// Mitsubishi GX Works2 project: PLC 특수기능 (연산 결과 반전)   PLC: Q03UDV

PROGRAM MAIN
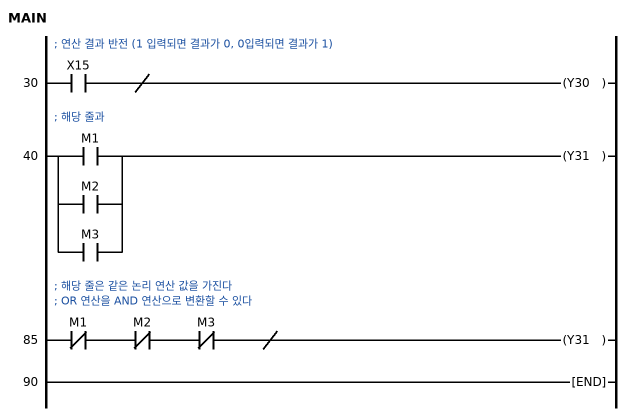
; 연산 결과 반전 (1 입력되면 결과가 0, 0입력되면 결과가 1)
30    LD      X15
      INV
      OUT     Y30
; 해당 줄과
40    LD      M1
      OR      M2
      OR      M3
      OUT     Y31
; 해당 줄은 같은 논리 연산 값을 가진다
; OR 연산을 AND 연산으로 변환할 수 있다
85    LDI     M1
      ANI     M2
      ANI     M3
      INV
      OUT     Y31
90    END
END_PROGRAM
